# B&R Automation Studio project AS-Lab-2-Chivin-AA-KRBO-03-18-main
Automation Studio 

## Logical view

### Program Logical/DoorCtrl

#### Variables.var
```iecst
VAR
	doorSM : FBGate := (0);
	ledSM : LedCtrl := (0);
	ETAD : UINT := 0;
	Speed : INT := 0;
	driveSM : DriveControl;
END_VAR
```

#### Main.cpp
```cpp
#include <bur/plctypes.h>

#ifdef _DEFAULT_INCLUDES
	#include <AsDefault.h>
#endif

// amount of memory to be allocated for heap storage must be specified for every ANSI C++ program with the bur_heap_size variable
unsigned long bur_heap_size = 0xFFFF;

void _INIT ProgramInit(void)
{
	driveSM.enable = 1;	// Insert code here

}

void _CYCLIC ProgramCyclic(void)
{
	FBGate (&doorSM);
	driveSM.speed=doorSM.speed;
	DriveControl(&driveSM);
	ledSM.state = doorSM.state;
	LedCtrl(&ledSM);
	L1=ledSM.s1;
	L2=ledSM.s2;
	L3=ledSM.s3;
	L4=ledSM.s4;
}

void _EXIT ProgramExit(void)
{
	// Insert code here

}
```

### Program Logical/LED

#### Variables.var
```iecst
VAR
	Led : LedCtrl;
	Led1 : BOOL;
	Led2 : BOOL;
	Led3 : BOOL;
	Led4 : BOOL;
END_VAR
```

#### Main.cpp
```cpp
#include <bur/plctypes.h>

#ifdef _DEFAULT_INCLUDES
	#include <AsDefault.h>
#endif

// amount of memory to be allocated for heap storage must be specified for every ANSI C++ program with the bur_heap_size variable
unsigned long bur_heap_size = 0xFFFF;

void _INIT ProgramInit(void)
{
	// Insert code here

}

void _CYCLIC ProgramCyclic(void)
{
	LedCtrl(&Led);

		Led1 = L1;
		Led2 = L2;
		Led3 = L3;
		Led4 = L4;
}

void _EXIT ProgramExit(void)
{
	// Insert code here

}
```

### Library Logical/Libraries/GateCtrl (ANSIC)

#### Types.typ - Exported data types
```iecst
TYPE
	GateState :
		(
		ST_INIT := 0,
		ST_UNKNOWN := 1,
		ST_OPEN := 2,
		ST_CLOSE := 3,
		ST_ACC_POS := 4,
		ST_ACC_NEG := 5,
		ST_POS := 6,
		ST_NEG := 7,
		ST_DEC_POS := 8,
		ST_DEC_NEG := 9
		);
	drivecommand :
		(
		CMD_SWITCHED_ON := 7,
		CMD_DISABLE_VOLTAGE := 0,
		CMD_ENABLE := 15,
		CMD_SHUTDOWN := 6,
		STATE_READY := 33,
		STATE_DISABLED := 64,
		STATE_SWITCHED_ON := 35
		);
END_TYPE
```

#### FBGate.c
```c
#include <bur/plctypes.h>
#ifdef __cplusplus
	extern "C"
	{
#endif
	#include "GateCtrl.h"
#ifdef __cplusplus
	};
#endif
/* TODO: Add your comment here */
void FBGate(struct FBGate* inst)
{
	/*TODO: Add your code here*/
	switch(inst->state)
	{
		case ST_INIT:
			{
				if(inst->sw1==0 && inst->sw2==0 && inst->sw3==0 && inst->sw4==0)
					inst->state=ST_UNKNOWN;
				break;
			}
		case ST_UNKNOWN:
			{
				if(inst->direction==0 && inst->sw1!=inst->swo1)
					inst->state=ST_CLOSE;
				if(inst->direction==1 && inst->sw1!=inst->swo1)
					inst->state=ST_NEG;
				if(inst->direction==1 && inst->sw2!=inst->swo2)
					inst->state=ST_ACC_NEG;
				if(inst->direction==1 && inst->sw3!=inst->swo3)
					inst->state=ST_DEC_NEG;

				if(inst->direction==1 && inst->sw4!=inst->swo4)
					inst->state=ST_OPEN;
				if(inst->direction==0 && inst->sw4!=inst->swo4)
					inst->state=ST_POS;
				if(inst->direction==0 && inst->sw3!=inst->swo3)
					inst->state=ST_ACC_POS;
				if(inst->direction==0 && inst->sw2!=inst->swo2)
					inst->state=ST_DEC_POS;
				break;
			}
		case ST_CLOSE:
			{
				inst->speed = 0;
				if(inst->direction==1)
					inst->state=ST_NEG;
				break;
			}
		case ST_NEG:
			{
				inst->speed = -300;
				if(inst->direction==1 && inst->sw2!=inst->swo2)
					inst->state=ST_ACC_NEG;
				if(inst->direction==0)
					inst->state=ST_DEC_POS;
				break;

			}
		case ST_ACC_NEG:
			{
				inst->speed = -600;
				if(inst->direction==1 && inst->sw3!=inst->swo3)
					inst->state=ST_DEC_NEG;
				if(inst->direction==0)
					inst->state=ST_ACC_POS;
				break;
			}
		case ST_DEC_NEG:
			{

				inst->speed = -200;
				if(inst->direction==1 && inst->sw4!=inst->swo4)
					inst->state=ST_OPEN;
				if(inst->direction==0)
					inst->state=ST_POS;
				break;
			}

		case ST_OPEN:
			{
				inst->speed = 0;
				if(inst->direction==0)
					inst->state=ST_POS;
				break;
			}
		case ST_POS:
			{
				inst->speed = 200;
				if(inst->direction==0 && inst->sw3!=inst->swo3)
					inst->state=ST_ACC_POS;
				if(inst->direction==1)
					inst->state=ST_DEC_NEG;
				break;
			}
		case ST_ACC_POS:
			{
				inst->speed = 600;
				if(inst->direction==0 && inst->sw2!=inst->swo2)
					inst->state=ST_DEC_POS;
				if(inst->direction==1)
					inst->state=ST_ACC_NEG;
				break;
			}
		case ST_DEC_POS:
			{
				inst->speed = 200;
				if(inst->direction==0 && inst->sw1!=inst->swo1)
					inst->state=ST_CLOSE;
				if(inst->direction==1)
					inst->state=ST_NEG;

				break;
			}
	}
	inst->swo1 = inst->sw1;
	inst->swo2 = inst->sw2;
	inst->swo3 = inst->sw3;
	inst->swo4 = inst->sw4;
}
```

#### GateCtrl.fun - Exported functions and function blocks
```iecst
{REDUND_ERROR} {REDUND_UNREPLICABLE} FUNCTION_BLOCK FBGate (*TODO: Add your comment here*) (*$GROUP=User,$CAT=User,$GROUPICON=User.png,$CATICON=User.png*)
	VAR_INPUT
		state : {REDUND_UNREPLICABLE} GateState;
		sw1 : {REDUND_UNREPLICABLE} BOOL;
		sw2 : {REDUND_UNREPLICABLE} BOOL;
		sw3 : {REDUND_UNREPLICABLE} BOOL;
		sw4 : {REDUND_UNREPLICABLE} BOOL;
		direction : {REDUND_UNREPLICABLE} BOOL;
	END_VAR
	VAR_OUTPUT
		speed : {REDUND_UNREPLICABLE} INT;
	END_VAR
	VAR
		swo1 : {REDUND_UNREPLICABLE} USINT;
		swo2 : {REDUND_UNREPLICABLE} USINT;
		swo3 : {REDUND_UNREPLICABLE} USINT;
		swo4 : {REDUND_UNREPLICABLE} USINT;
	END_VAR
END_FUNCTION_BLOCK

{REDUND_ERROR} FUNCTION_BLOCK LedCtrl (*TODO: Add your comment here*) (*$GROUP=User,$CAT=User,$GROUPICON=User.png,$CATICON=User.png*)
	VAR_INPUT
		state : {REDUND_UNREPLICABLE} GateState;
	END_VAR
	VAR_OUTPUT
		s1 : {REDUND_UNREPLICABLE} BOOL;
		s2 : {REDUND_UNREPLICABLE} BOOL;
		s3 : {REDUND_UNREPLICABLE} BOOL;
		s4 : {REDUND_UNREPLICABLE} BOOL;
		timer : INT;
	END_VAR
END_FUNCTION_BLOCK

{REDUND_ERROR} {REDUND_UNREPLICABLE} FUNCTION_BLOCK DriveControl (*TODO: Add your comment here*) (*$GROUP=User,$CAT=User,$GROUPICON=User.png,$CATICON=User.png*)
	VAR_INPUT
		enable : {REDUND_UNREPLICABLE} BOOL;
		state : {REDUND_UNREPLICABLE} UINT;
	END_VAR
	VAR_OUTPUT
		speed : {REDUND_UNREPLICABLE} INT;
		command : {REDUND_UNREPLICABLE} UINT;
	END_VAR
END_FUNCTION_BLOCK
```

#### LedCtrl.c
```c
#include <bur/plctypes.h>
#ifdef __cplusplus
	extern "C"
	{
#endif
#include "GateCtrl.h"
#ifdef __cplusplus
	};
#endif
/* TODO: Add your comment here */
void LedCtrl(struct LedCtrl* inst)
{
	{
		/*TODO: Add your code here*/
		switch(inst->state)
		{
			case ST_INIT:
				{
					inst->s1 = 0 ;
					inst->s2 = 0 ;
					inst->s3 = 0 ;
					inst->s4 = 0 ;
					break;
				}
			case ST_UNKNOWN:
				{
					if(inst->timer%10==0)
					{
						inst->s1 = !inst->s1;
						inst->s2 = !inst->s2;
						inst->s3 =
							!inst->s3;
						inst->s4 = !inst->s4;
					}
					break;
				}
			case ST_CLOSE:
				{

					inst->s1 = 1;
					inst->s2 = 1;
					inst->s3 = 1;
					inst->s4 = 1;
					break;
				}
			case ST_NEG:
				{

					inst->s1 = 0;
					inst->s2 = 1;
					inst->s3 = 1;
					inst->s4 = 1;
					break;
				}
			case ST_ACC_NEG:
				{

					inst->s1 = 0;
					inst->s2 = 0;
					inst->s3 = 1;
					inst->s4 = 1;
					break;
				}
			case ST_DEC_NEG:
				{

					inst->s1 = 0;
					inst->s2 = 0;
					inst->s3 = 0;
					inst->s4 = 1;
					break;
				}

			case ST_OPEN:
				{

					inst->s1 = 0;
					inst->s2 = 0;
					inst->s3 = 0;
					inst->s4 = 0;
					break;
				}
			case ST_POS:
				{

					inst->s1 = 0;
					inst->s2 = 0;
					inst->s3 = 0;
					inst->s4 = 1;
					break;
				}
			case ST_ACC_POS:
				{

					inst->s1 = 0;
					inst->s2 = 0;
					inst->s3 = 1;
					inst->s4 = 1;
					break;
				}
			case ST_DEC_POS:
				{

					inst->s1 = 0;
					inst->s2 = 1;
					inst->s3 = 1;
					inst->s4 = 1;
					break;
				}
		}
	}
	inst->timer++;
}
```

#### DriveControl.c
```c
#include <bur/plctypes.h>
#ifdef __cplusplus
extern "C"
{
#endif
#include "GateCtrl.h"
#ifdef __cplusplus
};
#endif
void DriveControl (struct DriveControl* inst)
{
	UINT mask = inst->state & 0x6f;
	if(!inst->enable)
	{
		inst->command = CMD_SHUTDOWN;
	}
	else
	{
		switch (mask)
		{
			//Выключенный двигатель
			case STATE_DISABLED:
				inst->command = CMD_SHUTDOWN;
				break;
			//Готовый двигатель
			case STATE_READY:
				inst->command = CMD_ENABLE;
				break;
			//Включенный двигатель
			case STATE_SWITCHED_ON:
				inst->command = CMD_SWITCHED_ON;
				break;
		}
	}
}
```

Listed in the project but not available here: Logical/Libraries/GateCtrl/Constants.var
